// TwinCAT 3 PLC project EpicsComModule
// ProgramVersion: 3.1.0.8
// libraries:
//   Tc2_EtherCAT, * (Beckhoff Automation GmbH)
//   Tc2_Standard, * (Beckhoff Automation GmbH)
//   Tc2_System, * (Beckhoff Automation GmbH)
//   Tc2_TcpIp, * (Beckhoff Automation GmbH)
//   Tc2_Utilities, * (Beckhoff Automation GmbH)
//   Tc3_Interfaces, * (Beckhoff Automation GmbH)
//   Tc3_Module, * (Beckhoff Automation GmbH)
// project tree:
//   Data types/ DUT_AxisStatus_v0_01.TcDUT (not stored), E_ConnectionSteps.TcDUT (not stored), E_ServerSteps.TcDUT (not stored), DUT_ComSettings.TcDUT (not stored)
//   Global Variables/ Global_Variables.TcGVL (not stored)
//   / PlcTaskCom.TcTTO (not stored)
//   POUs/DUT_Support/ FB_Read_DUT_AxisStatus_v0_01.TcPOU (not stored)
//   POUs/ FB_ServerApplication.TcPOU (not stored), FB_ServerConnection.TcPOU (not stored), FB_Server.TcPOU, FB_StreamBufferToADSBuffer.TcPOU (not stored), FB_ValidCommand.TcPOU (not stored), FB_ADSBufferToStreamBuffer.TcPOU (not stored), MAIN.TcPOU (not stored), README.TcPOU (not stored)
//   POUs/Helper POUs/ CheckBounds.TcPOU (not stored), FB_FindChar.TcPOU (not stored), FB_FrameFifo.TcPOU, FB_LogFifo.TcPOU (not stored), F_RemoveBytesFromBuffer.TcPOU
//   POUs/Static Command support/ FB_GetStaticADR.TcPOU, FB_ParseStaticCommand.TcPOU, FB_ParseStringToSymInfo.TcPOU (not stored), FB_SetStaticADSPort.TcPOU, FB_SetStaticADR.TcPOU (not stored), FB_ParseCommandOption.TcPOU

// ---- POUs/FB_Server.TcPOU
///#########################################################
///FB that handles TCP/IP server and the client connections. The code is based on Beckhoff sample code. However changes and additions have been made to this code for the general purpose EPICS interface.
/// 
///
///	Library:		
///
///	Global Variables:
///	- EPICS_MAX_FRAME_SIZE					
///	- EPICS_ARRAY_DELIMITER					
///	- EPICS_COMMAND_DELIMITER
/// - PLCPRJ_BUFFER_SIZE				 
///
///	Data types:
///	
///	External functions:
///		- TC2_Standard lib
///		- Tc2_Utilities lib
///		- Tc2_System lib
///		
///###########################################################

FUNCTION_BLOCK FB_Server
VAR
	sVersion: STRING:='0.9.0';
END_VAR
VAR_INPUT
	sSrvNetID		: T_AmsNetID	:= '';(* TwinCAT TCP/IP server network address *)
	sLocalHost		: T_IPv4Addr 	:= '127.0.0.1';(* Own IP address! *)
	nLocalPort		: UDINT 		:= 0;(* Server port number *)
	bEnable			: BOOL 			:= FALSE;(* TRUE => enable server data exchange, FALSE => disable *)
	tReconnect 		: TIME 			:= T#3S;(* Reopen new listener socket after this time *)
	bLog			: BOOL 			:= FALSE;(* TRUE => Enable log message output, FALSE => Disable *)
	sPrefix			: STRING 		:= 'SERVER::';(* Log message description string (allows the identification of log message source) *)
END_VAR
VAR_OUTPUT
	bListening		: BOOL			:= FALSE;(* Listener socket state *)
	nAccepted		: UDINT			:= 0;(* Max. number of accepted client connections *)
END_VAR
VAR
	aApplications	: ARRAY[1..MAX_CLIENT_CONNECTIONS] OF FB_ServerApplication;(* Server application control function blocks *)
	aConnections	: ARRAY[1..MAX_CLIENT_CONNECTIONS] OF FB_ServerConnection := 
													[ 	(sPrefix := 'SERVER1::'), 
														(sPrefix := 'SERVER2::'), 
														(sPrefix := 'SERVER3::'), 
														(sPrefix := 'SERVER4::'), 
														(sPrefix := 'SERVER5::') ];(* Server connection/data exchange control function blocks *)
	aTx 			: ARRAY[1..MAX_CLIENT_CONNECTIONS] OF FB_FrameFifo;(* TX fifo *)
	aRx 			: ARRAY[1..MAX_CLIENT_CONNECTIONS] OF FB_FrameFifo;(* RX fifo *)
	aLog			: ARRAY[1..MAX_CLIENT_CONNECTIONS] OF FB_LogFifo;(* Listener log message fifo *)
	fbListen	 	: FB_SocketListen;
	fbClose			: FB_SocketClose;
	fbLog			: FB_LogFifo;
	fbListenTimer	: TON;
	bReset			: BOOL := FALSE;
	eStep			: E_ServerSteps;
	i				: UDINT;
END_VAR



CASE eStep OF
	eSERVER_STATE_IDLE:
		IF bEnable XOR bListening THEN
			IF bEnable THEN
				fbListenTimer( IN := TRUE );
				IF fbListenTimer.Q THEN
					fbListenTimer( IN := FALSE, PT := tReconnect );

					fbLog.Clear( sPrefix := sPrefix, bLog := bLog );(* Clear listener log fifo *)
					bReset := FALSE;

					eStep := eSERVER_STATE_LISTENER_OPEN_START;
				END_IF
			ELSE
				eStep := eSERVER_STATE_REMOTE_CLIENTS_CLOSE;
			END_IF
		ELSIF bListening THEN
			eStep := eSERVER_STATE_REMOTE_CLIENTS_COMM;
		ELSE
			fbListenTimer( IN := FALSE, PT := T#0S );
			bReset := FALSE;
		END_IF

	eSERVER_STATE_LISTENER_OPEN_START:
		fbListen(  bExecute := FALSE  );
		fbListen( 	sSrvNetID := sSrvNetID, 
					sLocalHost := sLocalHost, 
					nLocalPort := nLocalPort, 
					bExecute := TRUE );
		eStep := eSERVER_STATE_LISTENER_OPEN_WAIT;

	eSERVER_STATE_LISTENER_OPEN_WAIT:
		fbListen( bExecute := FALSE );
		IF NOT fbListen.bBusy THEN
			IF NOT fbListen.bError THEN
				bListening 	:= TRUE;
				fbLog.Message( sMessage := 'Listener socket opened!', hSocket := fbListen.hListener );
				eStep := eSERVER_STATE_IDLE;
			ELSE
				fbLog.Error( sMessage := 'FB_SocketListen()', nErrId := fbListen.nErrId );
				eStep := eSERVER_STATE_ERROR;
			END_IF
		END_IF		

	eSERVER_STATE_REMOTE_CLIENTS_COMM:
		eStep := eSERVER_STATE_IDLE;
		nAccepted := 0;

		FOR i:= 1 TO MAX_CLIENT_CONNECTIONS DO
			aApplications[i].nConnectionIndex:=i;
			aConnections[i]( fbTx := aTx[i], fbRx := aRx[i], fbLog := aLog[i],
							hListener := fbListen.hListener, bReset := bReset,
							sSrvNetID := sSrvNetID, bEnable := bEnable,	bLog := bLog ); 
			IF bReset THEN
				bReset := FALSE; 
				eStep := eSERVER_STATE_REMOTE_CLIENTS_CLOSE;
				EXIT;
			END_IF
			
			IF aConnections[i].bAccepted THEN
				aApplications[i]( fbTx := aTx[i], fbRx := aRx[i], fbLog := aLog[i]);
				nAccepted := nAccepted + 1;(* Count the number of connected remote clients *)
				aApplications[i].bReset:=FALSE;
			ELSE
					aApplications[i].bReset:=TRUE;
					aApplications[i]( fbTx := aTx[i], fbRx := aRx[i], fbLog := aLog[i]);
			END_IF
			

		END_FOR

	eSERVER_STATE_REMOTE_CLIENTS_CLOSE:
		nAccepted := 0;
		FOR i:= 1 TO MAX_CLIENT_CONNECTIONS DO
			(* Close all remote client (accepted) sockets *)
			aConnections[i]( fbTx := aTx[i], fbRx := aRx[i], fbLog := aLog[i],
							hListener := fbListen.hListener, bReset := bReset,
							sSrvNetID := sSrvNetID, bEnable := FALSE, bLog := bLog ); 
			IF aConnections[i].bAccepted THEN
				nAccepted := nAccepted + 1;(* Count the number of connected remote clients *)
			END_IF
		END_FOR
		
		(* Check if all remote client sockets are closed *)
		IF nAccepted = 0 THEN
			eStep := eSERVER_STATE_LISTENER_CLOSE_START; (* Close listener socket too *)
		END_IF

	eSERVER_STATE_LISTENER_CLOSE_START:
		fbLog.Message( sMessage := 'Closing listener socket!', hSocket := fbListen.hListener );
		fbClose( bExecute := FALSE );
		fbClose( sSrvNetID := sSrvNetID, hSocket := fbListen.hListener, bExecute:= TRUE );
		eStep := eSERVER_STATE_LISTENER_CLOSE_WAIT;

	eSERVER_STATE_LISTENER_CLOSE_WAIT:
		fbClose( bExecute := FALSE );
		IF NOT fbClose.bBusy THEN
			bListening := FALSE;
			nAccepted := 0;
			IF NOT fbClose.bError THEN
				eStep := eSERVER_STATE_IDLE;
			ELSE
				fbLog.Error( sMessage := 'FB_SocketClose(listener)', nErrId := fbListen.nErrID );
				eStep := eSERVER_STATE_ERROR;
			END_IF
		END_IF

	eSERVER_STATE_ERROR:
		IF bListening THEN
			eStep := eSERVER_STATE_REMOTE_CLIENTS_CLOSE;
		ELSE
			eStep := eSERVER_STATE_IDLE;
		END_IF

END_CASE

END_FUNCTION_BLOCK

// ---- POUs/Helper POUs/FB_FrameFifo.TcPOU
(* Tx (byte data) fifo control function block (Older where based on string format) *)
FUNCTION_BLOCK FB_FrameFifo
VAR
	sVersion: STRING:='0.9.0';
END_VAR
VAR_INPUT
	bLog		: BOOL			:= FALSE;(* TRUE => Enable log message output, FALSE => Disable *)
	sPrefix		: STRING		:= 'Unknown::';(* Log message description string (allows the identification of log message source) *)
	bPut		: POINTER TO ARRAY[0..EPICS_MAX_FRAME_SIZE] OF BYTE; (* Byte message to add (write) to the fifo *)
	bGet		: POINTER TO ARRAY[0..EPICS_MAX_FRAME_SIZE] OF BYTE; (* Byte message removed (read) from fifo *)
	nWriteCount : UDINT:=0;
	nReadBufferSize : UDINT:=0;
END_VAR
VAR_OUTPUT
	bOk			: BOOL; 	 	(* TRUE = New entry added or removed succesfully, FALSE = Fifo overflow or fifo empty *)
	nCount		: UDINT			:= 0;(* Number of fifo entries *)
	cbFree		: UDINT 		:= 0;(* Free buffer space *)
	nReadCount	: UDINT:=0;
END_VAR
VAR
	fbBuffer 	: FB_MemRingBuffer;(* Basic (lower level) string buffer control function block *)
	buffer		: ARRAY[-3..PLCPRJ_BUFFER_SIZE] OF BYTE;(* Internal buffer memory *)
	sPut		: T_MaxString;
	nMax: UDINT;
	spBufferString: POINTER TO STRING;
END_VAR



;

ACTION Clear:
(* Resets fifo = clears all data *)
fbBuffer.A_Reset( pBuffer:= ADR(buffer), cbBuffer:= SIZEOF(buffer),
				bOk=>bOk, nCount=>nCount );
cbFree := PLCPRJ_BUFFER_SIZE;(* Free buffer size *)
END_ACTION

ACTION AddTail:
(* Adds new fifo entry *)
fbBuffer.A_AddTail( pBuffer:= ADR(buffer),pWrite:=bPut,cbWrite:=nWriteCount,cbBuffer:= SIZEOF(buffer),
					 bOk=>bOk, nCount=>nCount );

IF bOk THEN
	cbFree := PLCPRJ_BUFFER_SIZE - fbBuffer.cbSize;(* Calculate the free buffer space *)
	IF bLog THEN(* Log message *)
		IF 	nWriteCount>50 THEN
			nMax:=50;
		ELSE
			nMax:=nWriteCount;
		END_IF
		sPut:='';
		memcpy(destAddr:=ADR(sPut[0]),srcAddr:=(bPut+nWriteCount-nMax),n:=nMax); //Copy byte data to string
		sPut[nMax]:=0; //Terminate string
		ADSLOGSTR( ADSLOG_MSGTYPE_HINT OR ADSLOG_MSGTYPE_LOG, CONCAT( ''(*sPrefix*), '"%s"' ),sPut );
	END_IF
END_IF
END_ACTION

ACTION RemoveHead:
(* Removes oldest fifo entry *)
//fbBuffer.A_RemoveHead( pBuffer:= ADR(buffer), cbBuffer:= SIZEOF(buffer), pRead:=bGet,
//						bOk=>bOk,cbReturn=>nReadCount, nCount=>nCount, cbRead:=nReadBufferSize);
fbBuffer.A_RemoveHead( pBuffer:= ADR(buffer), cbBuffer:= SIZEOF(buffer), pRead:=bGet,
						bOk=>bOk,cbReturn=>nReadCount, nCount=>nCount, cbRead:=nReadBufferSize);
						
						
						
IF bOk THEN
	cbFree := PLCPRJ_BUFFER_SIZE - fbBuffer.cbSize;(* Calculate the free buffer space *)
	//ADSLOGSTR( ADSLOG_MSGTYPE_HINT OR ADSLOG_MSGTYPE_LOG, CONCAT( 'Took bytes OK: ', '"%s"' ) ,UDINT_TO_STRING(ncount));
ELSE
	
	//ADSLOGSTR( ADSLOG_MSGTYPE_HINT OR ADSLOG_MSGTYPE_LOG, CONCAT( ''(*sPrefix*), '"%s"' ),'Took bytes Fail' );
END_IF
END_ACTION

END_FUNCTION_BLOCK

// ---- POUs/Helper POUs/F_RemoveBytesFromBuffer.TcPOU
FUNCTION F_RemoveBytesFromBuffer : BOOL
VAR
	sVersion: STRING:='0.9.0';
END_VAR
VAR_INPUT	
	nRemoveBytes:UDINT:=0;
END_VAR
VAR_IN_OUT
	byteCommandBuffer	:	ARRAY[0..PLCPRJ_BUFFER_SIZE] OF BYTE;//ADS input buffer
	nBytesInCommandBuffer:DINT:=0;
	nIndexEndOfCommand:DINT:=0;
END_VAR


VAR
	nCommandEndIndex: DINT;
	bRet: BOOL;
END_VAR

//Remove ADS command from buffer
bRet:=FALSE;
IF nRemoveBytes>0 AND (nRemoveBytes< PLCPRJ_BUFFER_SIZE-nRemoveBytes) THEN 
	MEMMOVE(srcAddr:=ADR(byteCommandBuffer[nRemoveBytes]),destAddr:=ADR(byteCommandBuffer[0]),n:= nBytesInCommandBuffer-nRemoveBytes); //remove ADSPORT command from buffer
	MEMSET(destAddr:=ADR(byteCommandBuffer[nBytesInCommandBuffer-nRemoveBytes]),fillByte:=0,n:=nRemoveBytes); //reset buffer
	nBytesInCommandBuffer:=nBytesInCommandBuffer-nRemoveBytes;
	nIndexEndOfCommand:=nIndexEndOfCommand-nRemoveBytes;	
	bRet:=TRUE;
END_IF
F_RemoveBytesFromBuffer:=bREt;
RETURN;

END_FUNCTION

// ---- POUs/Static Command support/FB_GetStaticADR.TcPOU
FUNCTION_BLOCK FB_GetStaticADR
VAR
	sVersion: STRING:='0.9.0';
END_VAR
VAR_INPUT
	bEnable:BOOL:=FALSE;
	nCommadStartIndex:INT:=0;
	nCommandEndIndex:INT:=0;	
END_VAR
VAR
	psCommandBufferString: POINTER TO STRING; //string to point into byte buffer	
	nQuestionSign: INT;
END_VAR

VAR_IN_OUT
	byteCommandBuffer	:	ARRAY[0..PLCPRJ_BUFFER_SIZE] OF BYTE;//ADS input buffer
	nBytesInCommandBuffer:DINT:=0;
	nIndexEndOfCommand:DINT:=0;
END_VAR

VAR_OUTPUT
	nErrorId: UDINT;
	bError:BOOL:=FALSE;
	sVariableName:STRING(255);
	sSubErrorString: STRING;
END_VAR

//Static command/option 1: Check if ADR option	
(*IF bEnable THEN
	bError:=FALSE;
	nErrorId:=0;	
	sSubErrorString:='';	
	sVariableName:='';		
	psCommandBufferString:=ADR(byteCommandBuffer);
	nQuestionSign:=len(STR:=EPICS_STATIC_COMMAND_ABS_ADRESS);
	IF 	byteCommandBuffer[len(STR:=EPICS_STATIC_COMMAND_ABS_ADRESS)]=EPICS_ASCII_QUESTIONMARK AND nQuestionSign>0 THEN
		sVariableName:=right(str:=left(str:=PSTRING_TO_STRING(psCommandBufferString),size:=nCommandEndIndex-1),SIZE:=(nCommandEndIndex-1)-nQuestionSign-1);
		IF NOT F_RemoveBytesFromBuffer_V1_00(nRemoveBytes:= nCommandEndIndex,byteCommandBuffer:=byteCommandBuffer,nBytesInCommandBuffer:=nBytesInCommandBuffer,nIndexEndOfCommand:=nIndexEndOfCommand) THEN 			
			bError:=TRUE;
			nErrorId:=312;
			sSubErrorString:='State 3: Failed to clear buffer (ADR).';	
		END_IF
	ELSE
		nErrorId:=313;
		bError:=TRUE;
		sSubErrorString:='State 3: Failed to parse ADR set command.';	
	END_IF		
END_IF*)

END_FUNCTION_BLOCK

// ---- POUs/Static Command support/FB_ParseStaticCommand.TcPOU
FUNCTION_BLOCK FB_ParseStaticCommand
VAR
	sVersion: STRING:='0.9.0';
END_VAR
VAR
	psCommandBufferString: POINTER TO STRING; //string to point into byte buffer		
	nEqualSign: INT;
	nQuestionMark: INT;
END_VAR

VAR_IN_OUT
	byteCommandBuffer	:	ARRAY[0..PLCPRJ_BUFFER_SIZE] OF BYTE;//ADS input buffer
	nBytesInCommandBuffer:DINT:=0;
	nIndexEndOfCommand:DINT:=0;
END_VAR

VAR_OUTPUT
	nErrorId: UDINT;
	bError:BOOL:=FALSE;
	sSubErrorString: STRING;
	sStaticCommand:STRING;
	sStaticValue:STRING;
	bReadCommand:BOOL:=FALSE;
	bWriteCommand:BOOL:=FALSE;
END_VAR

//Parse static command	
nErrorId:=0;
bError:=FALSE;
sStaticCommand:='';
sStaticValue:='';
bReadCommand:=FALSE;
bWriteCommand:=FALSE;
psCommandBufferString:=ADR(byteCommandBuffer);

nEqualSign:=find(STR1:=PSTRING_TO_STRING(psCommandBufferString),STR2:=EPICS_WRITE_CMD);	
IF nEqualSign>0 AND nEqualSign<=nIndexEndOfCommand THEN
	bWriteCommand:=TRUE;	
	//Command
	memcpy(destAddr:=ADR(sStaticCommand[0]),srcAddr:=ADR(byteCommandBuffer[0]),n:=nEqualSign-1);
	memset(destAddr	:=ADR(sStaticCommand[nEqualSign-1]),fillByte:=0,n:=1);				//Terminate string	
	//Value
	memcpy(destAddr:=ADR(sStaticValue[0]),srcAddr:=ADR(byteCommandBuffer[nEqualSign]),n:=nIndexEndOfCommand-nEqualSign-1);
	memset(destAddr	:=ADR(sStaticValue[nIndexEndOfCommand-nEqualSign-1]),fillByte:=0,n:=1); //Terminate string
	IF NOT F_RemoveBytesFromBuffer_V1_00(nRemoveBytes:= nIndexEndOfCommand,byteCommandBuffer:=byteCommandBuffer,nBytesInCommandBuffer:=nBytesInCommandBuffer,nIndexEndOfCommand:=nIndexEndOfCommand) THEN 			
		bError:=TRUE;
		nErrorId:=301;
		sSubErrorString:='State 3: Failed to clear buffer (Parse static command write).';	
	END_IF				
ELSE
	nQuestionMark:=find(STR1:=PSTRING_TO_STRING(psCommandBufferString),STR2:=EPICS_READ_CMD);	
	IF nQuestionMark>0 AND nQuestionMark<=nIndexEndOfCommand THEN
		bReadCommand:=TRUE;	
		//Command
		memcpy(destAddr:=ADR(sStaticCommand[0]),srcAddr:=ADR(byteCommandBuffer[0]),n:=nQuestionMark-1);
		memset(destAddr	:=ADR(sStaticCommand[nQuestionMark-1]),fillByte:=0,n:=1);				//Terminate string	

		//Clean buffer
		IF NOT F_RemoveBytesFromBuffer_V1_00(nRemoveBytes:= nIndexEndOfCommand,byteCommandBuffer:=byteCommandBuffer,nBytesInCommandBuffer:=nBytesInCommandBuffer,nIndexEndOfCommand:=nIndexEndOfCommand) THEN 			
			bError:=TRUE;
			nErrorId:=302;
			sSubErrorString:='State 3: Failed to clear buffer (Parse static command read).';	
		END_IF		
	END_IF
END_IF	

IF NOT (bReadCommand OR  bWriteCommand) THEN										
	bError:=TRUE;
	nErrorId:=303;
	sSubErrorString:='State 3: Parsing of static command failed.';	
END_IF

END_FUNCTION_BLOCK

// ---- POUs/Static Command support/FB_SetStaticADSPort.TcPOU
FUNCTION_BLOCK FB_SetStaticADSPort
VAR
	sVersion: STRING:='0.9.0';
END_VAR
VAR_INPUT
	bEnable:BOOL:=FALSE;
	nCommadStartIndex:INT:=0;
	nCommandEndIndex:INT:=0;	
END_VAR
VAR
	psCommandBufferString: POINTER TO STRING; //string to point into byte buffer	
	bInStaticSection: BOOL;	
	sTemp: STRING;
	nEqualSign: INT;
END_VAR

VAR_IN_OUT
	byteCommandBuffer	:	ARRAY[0..PLCPRJ_BUFFER_SIZE] OF BYTE;//ADS input buffer
	nBytesInCommandBuffer:DINT:=0;
	nIndexEndOfCommand:DINT:=0;
END_VAR

VAR_OUTPUT
	nErrorId: UDINT;
	bError:BOOL:=FALSE;
	nADSPort: UINT:=0;
	sSubErrorString: STRING;
END_VAR

//Static command/option 1: Check if ADSPORT option	
IF bEnable THEN
	psCommandBufferString:=ADR(byteCommandBuffer);
	nEqualSign:=find(STR1:=PSTRING_TO_STRING(psCommandBufferString),STR2:=EPICS_WRITE_CMD);															
	sTemp:=right(str:=left(str:=PSTRING_TO_STRING(psCommandBufferString),size:=nCommandEndIndex-1),SIZE:=(nCommandEndIndex-1)-nEqualSign);
	nADSPort:=STRING_TO_UINT(sTemp);	
	IF nADSPort<1 OR nADSPort>20000 THEN
		nErrorId:=301;
		bError:=TRUE;
		sSubErrorString:='State 3: ADSPORT out of range.';
	//	nADSPort:=EPICS_ADS_PORT; //Set to default
	END_IF						
	//Remove ADS command from buffer
	IF NOT F_RemoveBytesFromBuffer_V1_00(nRemoveBytes:= nCommandEndIndex,byteCommandBuffer:=byteCommandBuffer,nBytesInCommandBuffer:=nBytesInCommandBuffer,nIndexEndOfCommand:=nIndexEndOfCommand) THEN 			
			bError:=TRUE;
			nErrorId:=302;
			sSubErrorString:='State 3: Failed to clear buffer (ADSPORT)).';	
	END_IF							
END_IF

END_FUNCTION_BLOCK

// ---- POUs/Static Command support/FB_ParseCommandOption.TcPOU
FUNCTION_BLOCK FB_ParseCommandOption
VAR
	sVersion: STRING:='0.9.0';
END_VAR
VAR_INPUT
	nCommandEndIndex:INT:=0;	
END_VAR
VAR
	psCommandBufferString: POINTER TO STRING; //string to point into byte buffer		
	nEqualSign: INT;
	nQuestionMark: INT;
END_VAR

VAR_IN_OUT
	byteCommandBuffer	:	ARRAY[0..PLCPRJ_BUFFER_SIZE] OF BYTE;//ADS input buffer
	nBytesInCommandBuffer:DINT:=0;
	nIndexEndOfCommand:DINT:=0;
END_VAR

VAR_OUTPUT
	nErrorId: UDINT;
	bError:BOOL:=FALSE;
	sSubErrorString: STRING;
	sStaticCommand:STRING;
	sStaticValue:STRING;
	bReadCommand:BOOL:=FALSE;
	bWriteCommand:BOOL:=FALSE;
	bWritePersistent:BOOL:=FALSE;	
END_VAR

//Parse static command	
nErrorId:=0;
bError:=FALSE;
sStaticCommand:='';
sStaticValue:='';
bReadCommand:=FALSE;
bWriteCommand:=FALSE;
bWritePersistent:=FALSE;		
psCommandBufferString:=ADR(byteCommandBuffer);

nEqualSign:=find(STR1:=PSTRING_TO_STRING(psCommandBufferString),STR2:=EPICS_WRITE_CMD);	
IF nEqualSign>0 AND nEqualSign<nCommandEndIndex THEN
	bWriteCommand:=TRUE;	
	//Command
	memcpy(destAddr:=ADR(sStaticCommand[0]),srcAddr:=ADR(byteCommandBuffer[0]),n:=nEqualSign-1);
	memset(destAddr	:=ADR(sStaticCommand[nEqualSign-1]),fillByte:=0,n:=1);				//Terminate string	
	//Check if persistent
	//IF find(STR1:=sStaticCommand,STR2:=EPICS_STATIC_COMMAND_PERSISTENT)>0 THEN
//		bWritePersistent:=TRUE;
//	END_IF
	//Value
	memcpy(destAddr:=ADR(sStaticValue[0]),srcAddr:=ADR(byteCommandBuffer[nEqualSign]),n:=nCommandEndIndex-nEqualSign-1);
	memset(destAddr	:=ADR(sStaticValue[nCommandEndIndex-nEqualSign-1]),fillByte:=0,n:=1); //Terminate string
	IF NOT F_RemoveBytesFromBuffer(nRemoveBytes:= nCommandEndIndex,byteCommandBuffer:=byteCommandBuffer,nBytesInCommandBuffer:=nBytesInCommandBuffer,nIndexEndOfCommand:=nIndexEndOfCommand) THEN 			
		bError:=TRUE;
		nErrorId:=301;
		sSubErrorString:='State 3: Failed to clear buffer (Parse static command write).';	
	END_IF				
ELSE
	nQuestionMark:=find(STR1:=PSTRING_TO_STRING(psCommandBufferString),STR2:=EPICS_READ_CMD);	
	IF nQuestionMark>0 AND nQuestionMark<nCommandEndIndex THEN
		bReadCommand:=TRUE;	
		//Command
		memcpy(destAddr:=ADR(sStaticCommand[0]),srcAddr:=ADR(byteCommandBuffer[0]),n:=nQuestionMark-1);
		memset(destAddr	:=ADR(sStaticCommand[nQuestionMark-1]),fillByte:=0,n:=1);				//Terminate string	

		//Clean buffer
		IF NOT F_RemoveBytesFromBuffer(nRemoveBytes:= nCommandEndIndex,byteCommandBuffer:=byteCommandBuffer,nBytesInCommandBuffer:=nBytesInCommandBuffer,nIndexEndOfCommand:=nIndexEndOfCommand) THEN 			
			bError:=TRUE;
			nErrorId:=302;
			sSubErrorString:='State 3: Failed to clear buffer (Parse static command read).';	
		END_IF		
	END_IF
END_IF	

IF NOT (bReadCommand OR  bWriteCommand) THEN										
	bError:=TRUE;
	nErrorId:=303;
	sSubErrorString:='State 3: Parsing of static command failed).';	
END_IF

END_FUNCTION_BLOCK
